{attribute 'qualified_only'}
{attribute 'to_string'}
TYPE E_GCSingleProcessResult :
(
	None := 0,
	Running := 1,
	Completed := 2,
	Stopped := 3,
	Aborted := 4,
	Failed := 5
) UINT;
END_TYPE

(* stored: Version 1.1.0.1, ProductVersion 3.1.4026.18
   DUT E_GCSingleProcessResult: Id {29e082ec-d45f-428f-911f-a33396d423b9} *)
